// A body that takes several scans, like most real tests.

//

// Returns FALSE until it has been called ScansToTake times, then records one check

// and returns TRUE. Counts its calls so the runner can be held to calling it

// exactly that many times - no more, no fewer.
FUNCTION_BLOCK SpanningTest IMPLEMENTS I_Test
VAR
	_ScansToTake	   : UDINT := 3;
	_BodyCalls		   : UDINT;
	_AbandonCalls	   : UDINT;
	_FirstCycleAtStart : BOOL;
	_CyclesAtFinish	   : UDINT;
	_Seen			   : BOOL;
END_VAR

// Calls received with Enable FALSE. Exactly one after an abandon.
PROPERTY AbandonCalls : UDINT
GET
AbandonCalls := _AbandonCalls;
END_GET
END_PROPERTY

PROPERTY BodyCalls : UDINT
GET
BodyCalls := _BodyCalls;
END_GET
END_PROPERTY

// ElapsedCycles the body saw on its last call. Counts the BODY only, not setup.
PROPERTY CyclesAtFinish : UDINT
GET
CyclesAtFinish := _CyclesAtFinish;
END_GET
END_PROPERTY

// I_TestTiming.IsFirstCycle as the body saw it on its first call. TRUE even when

// setup consumed scans first - the body's first scan is the body's first scan.
PROPERTY FirstCycleAtStart : BOOL
GET
FirstCycleAtStart := _FirstCycleAtStart;
END_GET
END_PROPERTY

METHOD Run : BOOL
VAR_INPUT
	Enable : BOOL;
	Test   : I_TestAssertions;
END_VAR
IF NOT Enable THEN
	_AbandonCalls := _AbandonCalls + 1;
	Run			  := TRUE;
	RETURN;
END_IF

_BodyCalls := _BodyCalls + 1;
IF NOT _Seen THEN
	// Captured on the body's FIRST call, whatever setup did beforehand.
	_Seen			   := TRUE;
	_FirstCycleAtStart := Test.IsFirstCycle;
END_IF

IF _BodyCalls < _ScansToTake THEN
	Run := FALSE;
	RETURN;
END_IF

_CyclesAtFinish := Test.ElapsedCycles;
Test.AssertTrue(TRUE, 'reached the end');
Run := TRUE;
END_METHOD

// How many scans the body should take before finishing.
METHOD SetScans
VAR_INPUT
	Scans : UDINT;
END_VAR
_ScansToTake := Scans;
END_METHOD

END_FUNCTION_BLOCK

(* stored: Version 1.1.0.1, ProductVersion 3.1.4026.18
   POU SpanningTest: Id {0c22d57b-bebe-4586-ba98-f0f3cc602640}, SpecialFunc None
   Folder I_Test: Id {d035bd5b-64f5-4af4-8696-4769b9fcc1a5}
   Property AbandonCalls: Id {d92ad1e9-bb64-4d3e-9817-befd5ee50907}
   Get Get: Id {606305d8-1933-4952-a542-78ce8cf88a34}
   Property BodyCalls: Id {91af80d5-d9d8-4102-9091-0913fe4a63f8}
   Get Get: Id {4192bd92-7c93-40e2-8b9f-b23497a5f508}
   Property CyclesAtFinish: Id {da69fc5a-2ef9-41f0-8898-9853c0dc2049}
   Get Get: Id {03c70270-49bb-4bd7-ae14-c9ddae5a8dcf}
   Property FirstCycleAtStart: Id {51d793a7-4863-4430-a8a3-6484e819ec95}
   Get Get: Id {b9109e60-e1cb-453b-b06e-07f3a34cf415}
   Method Run: Id {ec287a6b-8ab4-439b-8b6d-c08175d95b72}
   Method SetScans: Id {248a0030-e074-4c15-95af-248d5b68704c} *)
